(*********************************** G.D S.p.A. - Technical Department ***********************************
============= PROGRAM INFO ============
FOLDER:             TBD
MACHINES INVOLVED:  TBD 

============= DESCRIPTION =============
csp machine declaration

============= REVISIONS ===============
Date		Version	 	Author      	Description             
----------	-------		------------  	--------------------------------------------
2019/04/05 	0000.00	 	M.Grasso		Creation of the PRG

**********************************************************************************************************)
(*$R process_ref := prc; $*)
PROGRAM csp_case_flapControl_os
VAR
	
	prc:											process;
	prc_path:										STRING;
	
END_VAR

_read_var_input();

_object_manager();

IF NOT objects_running()
THEN
	RETURN;	
END_IF

_read_process_image();

_mode_manager();

_set_runtime_properties();

(********************************* BODY *********************************)
(************************************************************************)

_handle_messages();

_write_output();

ACTION _handle_messages:
;
END_ACTION

ACTION _handle_process_test:
;
END_ACTION

ACTION _mode_manager:
IF process_mode_req_is_pending(prc)
THEN
    process_apply_mode_req_first_step(prc);
    CASE process_get_mode(prc) OF
        MODE_TO_ABSENT:
			;
        MODE_TO_INACTIVE:
			;
        MODE_TO_TEST:
			;
        MODE_TO_OPERATIONAL:
			;
    END_CASE
    process_apply_mode_req_second_step(prc);
END_IF
END_ACTION

ACTION _object_manager:
IF objects_initialization()
THEN
	sub_process_init(
		object_name					:= 'csp_case_flapControl_os.prc', 
		process						:= csp_case_flapControl.prc, 
		CONVERSION_this				:= prc);
		
	prc_path 						:= process_get_path(prc);
END_IF

IF objects_running()
THEN
	process_cycle(prc);
END_IF
END_ACTION

ACTION _read_process_image:
;
END_ACTION

ACTION _read_var_input:
;
END_ACTION

ACTION _set_runtime_properties:
;
END_ACTION

ACTION _write_output:
;
END_ACTION

END_PROGRAM

(* stored: Version 1.1.0.1, ProductVersion 3.1.4022.12
   POU csp_case_flapControl_os: Id {18190f33-4b1f-45d0-9d65-de454a054061}, SpecialFunc None
   Action _handle_messages: Id {9fce3b0a-70e7-497d-9b83-676099ded738}
   Action _handle_process_test: Id {b8c7a230-c1f1-4a4f-a7a9-663e2b944f77}
   Action _mode_manager: Id {12cd9dd5-58cd-4c49-904e-ab285531e7c6}
   Action _object_manager: Id {f2318e51-e058-43e0-9a1c-df057541714e}
   Action _read_process_image: Id {293d3003-1dd2-44ba-aaca-22f566f4d7d0}
   Action _read_var_input: Id {76a82347-b22c-4d0e-9c85-e91612ddc1ff}
   Action _set_runtime_properties: Id {b6eb7d52-33bc-4ccd-a404-8205511ce13b}
   Action _write_output: Id {9095836f-f9b3-4061-9000-bf6bdd37b1f0} *)
